TYPE ST_ROTATION_MOTOR :
STRUCT
	CURRENT_STATUS:DINT;
	CURRENT_PV:REAL;
	CURRENT_SET_PV:DINT;
	
	SET_CONTROL_VALUE:REAL;
	SET_PRESSURE:DINT;
	SET_CONTROL_MODE:DINT;
END_STRUCT
END_TYPE

(* stored: Version 1.1.0.1, ProductVersion 3.1.4024.12
   DUT ST_ROTATION_MOTOR: Id {8f21ebf1-de96-4041-af96-ebe243217a37} *)
